// TIA Portal V18 export
// export: Created 2026-06-09T02:36:17.7425322Z, ExportSetting WithDefaults, DisplayName Totally Integrated Automation Portal, DisplayVersion V18, DisplayName TIA Portal Openness, DisplayVersion V18, DisplayName TIA Portal Version Control Interface, DisplayVersion V18, DisplayName STEP 7 Professional, DisplayVersion V18, DisplayName STEP 7 Safety, DisplayVersion V18, DisplayName WinCC Professional, DisplayVersion V18
VAR_GLOBAL   // PLC tag table "Standard-Variablentabelle"
   Tag_1 AT %Q0.0 : Bool;
   Tag_2 AT %I0.0 : Bool;
   Tag_3 AT %I0.1 : Bool;
   "Warning Light" AT %Q1.2 : Bool;
END_VAR
